FUNCTION_BLOCK CORNERHARRIS (* openCV CornerHarris *)
  (* Version 1.0, AN, SWDC RTSoft *)
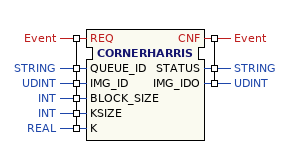
  EVENT_INPUT
    REQ WITH QUEUE_ID, IMG_ID, BLOCK_SIZE, KSIZE, K;
  END_EVENT
  EVENT_OUTPUT
    CNF WITH STATUS, IMG_IDO;
  END_EVENT
  VAR_INPUT
    QUEUE_ID : STRING;
    IMG_ID : UDINT;
    BLOCK_SIZE : INT; (* Neighborhood size *)
    KSIZE : INT; (* Aperture parameter for the Sobel operator *)
    K : REAL; (* Harris detector free parameter *)
  END_VAR
  VAR_OUTPUT
    STATUS : STRING;
    IMG_IDO : UDINT;
  END_VAR
  ALGORITHM REQ IN ST:

  END_ALGORITHM
END_FUNCTION_BLOCK
